PROGRAM S04_AluCovering
VAR
	//工站
	station					: REFERENCE TO FB_Station:=fbstation[4];
	//气缸
	fbHOZAdjustCyl_1	:REFERENCE TO FB_Cylinder:=fbCylinder[20];	//	上层水平调整气缸1
	fbHOZAdjustCyl_2	:REFERENCE TO FB_Cylinder:=fbCylinder[21];	//	上层水平调整气缸2
	fbHOZAdjustCyl_3	:REFERENCE TO FB_Cylinder:=fbCylinder[22];	//	下层水平调整气缸1
	fbHOZAdjustCyl_4	:REFERENCE TO FB_Cylinder:=fbCylinder[23];	//	下层水平调整气缸2
	//伺服
	fbZAxisMove_1	 :REFERENCE TO FB_Axis:=fbAxis[10];	//	热熔工位-Z轴伺服1（右）
	fbZAxisMove_2	 :REFERENCE TO FB_Axis:=fbAxis[11];	//		热熔工位-Z轴伺服2
	//温控器
	fbThermostat_1			 :REFERENCE TO FB_TempControl_FUSHI:=fbTempretureControl[1];//温控器1
    fbThermostat_2			 :REFERENCE TO FB_TempControl_FUSHI:=fbTempretureControl[2];//温控器2
	//延时
	arTonDelay :ARRAY[1..20] OF TON;
	//返回值
	UdiReturnValue :ARRAY[1..20] OF UDINT;
	//本地过程数据
	arProcessDataStation : ARRAY [1..2] OF DUT_MainlineFixture;
	i: INT;
	//过程记录
	tsModuleProcess:ARRAY[1..gc_ModuleProNo] OF DUT_Process;
	xClearModuleProcessDone:BOOL;
	bClearProcessStep	:BYTE;
END_VAR

ACTION A_Input:
//气缸
fbHOZAdjustCyl_1.xWP_Sensor	:=	IxS04HOZAdjustCyl_1WP	;
fbHOZAdjustCyl_1.xHP_Sensor	:=	IxS04HOZAdjustCyl_1HP	;
fbHOZAdjustCyl_2.xWP_Sensor	:=	IxS04HOZAdjustCyl_2WP	;
fbHOZAdjustCyl_2.xHP_Sensor	:=	IxS04HOZAdjustCyl_2HP	;
fbHOZAdjustCyl_3.xWP_Sensor	:=	IxS04HOZAdjustCyl_3WP	;
fbHOZAdjustCyl_3.xHP_Sensor	:=	IxS04HOZAdjustCyl_3HP	;
fbHOZAdjustCyl_4.xWP_Sensor	:=	IxS04HOZAdjustCyl_4WP	;
fbHOZAdjustCyl_4.xHP_Sensor	:=	IxS04HOZAdjustCyl_4HP	;
END_ACTION

ACTION Alarm:
//
station.adwAlarm[1].00:=station.xInitTimeout;	  			//S08Label 初始化超时
END_ACTION

ACTION Delay:
(*arTonDelay[01](IN:= , PT:=T#0.1S , Q=> , ET=> );*)//TipAuto使用
arTonDelay[02](IN:=  , PT:=stData.Thermostat[1].tTON_Delay , Q=> , ET=> );//热熔延时时间
arTonDelay[03](IN:=   , PT:=T#1S , Q=> , ET=> );
arTonDelay[04](IN:= , PT:=T#0.1S , Q=> , ET=> );
arTonDelay[05](IN:= , PT:=T#0.1S , Q=> , ET=> );
arTonDelay[06](IN:= , PT:=T#0.1S , Q=> , ET=> );
arTonDelay[07](IN:= , PT:=T#0.1S , Q=> , ET=> );
arTonDelay[08](IN:= , PT:=T#0.1S , Q=> , ET=> );
arTonDelay[09](IN:= , PT:=T#0.1S , Q=> , ET=> );
END_ACTION

ACTION FlowAuto:

//-----------------------------------------初始化是否完成判断----------------------------------------------
IF NOT station.xInitDone 
THEN
 	station.iStepAuto:=0;
 	station.xDone:=FALSE;
	station.xRunningOffProhibit := FALSE ;//运行中信号Off禁止
ELSIF station.xRunning  OR   tsModuleProcess[2].xProcessStarted
THEN
//-----------------------------------------动作步骤--------------------------------------------------------
CASE station.iStepAuto OF	  
	0: //----Home Step，等待启动----
		IF station.xDisabled 
			AND station.xCanRun 
			AND NOT fbMachine[1].xStopped 
			AND NOT station.xSingleRunning 
		THEN
			station.xDone:=TRUE;
		END_IF
		
		IF  station.xSingleRunning 
			OR station.xCanRun 
			AND NOT station.xDone 
			AND NOT station.xDisabled 
			AND NOT fbMachine[1].xStopped
		THEN
			station.xCycleEnable:=TRUE;
			station.xDone:= FALSE;  
			station.xRunningOffProhibit := TRUE ;//运行中信号Off禁止
			station.iStepAuto:= 10;
		END_IF
    10: //复位数据
			(*开启控温系统*) 
			fbThermostat_1.xStart :=TRUE;
			fbThermostat_2.xStart :=TRUE;
			arTonDelay[02](IN:= FALSE);
			station.iStepAuto:=20;	
	20:////Restore_after_Estop_Process1 上载数据流程
			IF  station.xSingleRunning OR  fbMachine[1].xTryRun THEN
					station.iStepAuto:=50;
			ELSIF tsModuleProcess[1].xProcessNotStarted AND NOT  tsModuleProcess[1].xProcessStarted THEN
					station.iStepAuto :=21; (*process not started*)
			ELSIF  tsModuleProcess[1].xProcessStarted AND NOT  tsModuleProcess[1].xProcessCompleted THEN
				 station.iStepAuto := 21;(*process started*)
			ELSIF  tsModuleProcess[1].xProcessCompleted AND NOT tsModuleProcess[1].xQDataCompleted  THEN
					station.iStepAuto := 40 ;(*process completed*)
			ELSIF tsModuleProcess[1].xQDataCompleted THEN
					station.iStepAuto :=40;(*Qdata completed *)
			ELSE
					station.iStepAuto :=21; 
			END_IF	
	21://
				tsModuleProcess[1].xProcessNotStarted:=TRUE;
				station.iStepAuto:= 30;
				
	30://数据load 
		tsModuleProcess[1].xProcessStarted	:=TRUE;
		MEMCPY(ADR(arProcessDataStation[1]),ADR(arMainlineFixtureData[arCurFixtureNumStation[10]]),SIZEOF(arMainlineFixtureData[arCurFixtureNumStation[10]]));
		MEMCPY(ADR(arProcessDataStation[2]),ADR(arMainlineFixtureData[arCurFixtureNumStation[11]]),SIZEOF(arMainlineFixtureData[arCurFixtureNumStation[11]]));
		tsModuleProcess[1].xProcessCompleted:=TRUE;
		tsModuleProcess[1].xQDataCompleted:=TRUE;
		station.iStepAuto:= 40;
	40: //判断产品状态
			IF  arProcessDataStation[1].xMaterialOnOff   AND
				 arProcessDataStation[2].xMaterialOnOff  THEN
				station.iStepAuto:= 41;
			ELSE
				station.iStepAuto:= 999;
			END_IF
	41://手动NOK按钮
			IF   arManualNOKHmiButton[4]  AND NOT station.xCycleRunning THEN
				station.iStepAuto:= 140;
			ELSE	
				station.iStepAuto:= 50;
			END_IF	
	
	/////产品流程开始	
	50:////Restore_after_Estop_Process2 热熔流程
			IF  station.xSingleRunning OR fbMachine[1].xTryRun THEN
					station.iStepAuto :=60; 
			ELSIF tsModuleProcess[2].xProcessNotStarted AND NOT  tsModuleProcess[2].xProcessStarted THEN
					station.iStepAuto :=60; (*process not started*)
			ELSIF  tsModuleProcess[2].xProcessStarted AND NOT  tsModuleProcess[2].xProcessCompleted THEN
				 station.iStepAuto := 140;(*process started*)
			ELSIF  tsModuleProcess[2].xProcessCompleted AND NOT tsModuleProcess[2].xQDataCompleted  THEN
					station.iStepAuto :=130;(*process completed*)
			ELSIF tsModuleProcess[2].xQDataCompleted THEN
					station.iStepAuto :=160;(*Qdata completed *)
			ELSE
					station.iStepAuto :=60; 
			END_IF	
	60://
				 tsModuleProcess[2].xProcessNotStarted:=TRUE;
				 station.iStepAuto :=70; 
	70://水平调整气缸伸出
					IF  iBoxChoose =1 THEN
						(*上层水平调整气缸*)
						fbHOZAdjustCyl_1.xAuto :=TRUE;
						fbHOZAdjustCyl_2.xAuto :=TRUE;
						IF  fbHOZAdjustCyl_1.xWP_Delay AND fbHOZAdjustCyl_2.xWP_Delay  THEN
								station.iStepAuto:= 80;
						END_IF
					ELSIF  iBoxChoose= 2 THEN
						(*下层水平调整气缸*)
						fbHOZAdjustCyl_3.xAuto :=TRUE;
						fbHOZAdjustCyl_4.xAuto :=TRUE;
						IF  fbHOZAdjustCyl_3.xWP_Delay AND fbHOZAdjustCyl_4.xWP_Delay  THEN
								station.iStepAuto:= 80;
						END_IF
					END_IF
	
	80://判断加热棒是否准备就绪
			IF  ( fbThermostat_1.xRdy AND  fbThermostat_2.xRdy ) OR 
				axBypassSignal[4] OR  fbMachine[1].xTryRun THEN
					station.iStepAuto:= 90;
			END_IF
	90://Z轴伺服下降到位置1
			tsModuleProcess[2].xProcessStarted:=TRUE;
			fbZAxisMove_1.xMoveAuto[2]:=TRUE;
			fbZAxisMove_2.xMoveAuto[2]:=TRUE;
			IF  fbZAxisMove_1.xMoveInPos[2] AND fbZAxisMove_2.xMoveInPos[2]THEN
				station.iStepInit:=100;	
			END_IF
	100://复位热熔时间
			arTonDelay[02](IN:=FALSE  , PT:=stData.Thermostat[1].tTON_Delay , Q=> , ET=> );//热熔延时时间
			station.iStepAuto:=110;
 	110://延时等待热熔完成
			arTonDelay[02](IN:=  , PT:=stData.Thermostat[1].tTON_Delay , Q=> , ET=> );//热熔延时时间
		IF  arTonDelay[02].Q  OR axBypassSignal[4]  OR fbMachine[1].xTryRun  THEN
			station.iStepInit:=120;	
			arTonDelay[02](IN:= FALSE );//热熔延时时间
		END_IF
	120://
			tsModuleProcess[2].xProcessCompleted :=TRUE;
			station.iStepInit:=130;	
	130://结果OK
			arProcessDataStation[1].stProduct.xAluCovering_NOK:=TRUE;
			arProcessDataStation[2].stProduct.xAluCovering_OK:=FALSE;
			station.iStepInit:=150;	
	140://结果NG 
			arProcessDataStation[1].stProduct.xAluCovering_NOK:=FALSE;
			arProcessDataStation[2].stProduct.xAluCovering_OK:=TRUE;		
			station.iStepInit:=150;	
	150:
			tsModuleProcess[2].xQDataCompleted :=TRUE;
			station.iStepInit:=160;	
	160://Z轴上升
			fbZAxisMove_1.xMoveAuto[1]:=TRUE;
			fbZAxisMove_2.xMoveAuto[1]:=TRUE;
			IF  fbZAxisMove_1.xMoveInPos[1] AND fbZAxisMove_2.xMoveInPos[1]THEN
				station.iStepInit:=170;	
			END_IF
	170://水平调整气缸收回
			fbHOZAdjustCyl_1.xAuto :=FALSE;
			fbHOZAdjustCyl_2.xAuto :=false;
			fbHOZAdjustCyl_3.xAuto :=false;
			fbHOZAdjustCyl_4.xAuto :=false;
		IF	fbHOZAdjustCyl_1.xhp_Delay AND
		    fbHOZAdjustCyl_2.xhp_Delay and
		    fbHOZAdjustCyl_3.xhp_Delay and
		    fbHOZAdjustCyl_4.xhp_Delay THEN
			station.iStepInit:=200;	
		END_IF
	////产品流程结束	
	200:////Restore_after_Estop_Process3 数据传输流程
			IF  station.xSingleRunning OR fbMachine[1].xTryRun THEN
					station.iStepAuto :=999; 
			ELSIF tsModuleProcess[3].xProcessNotStarted AND NOT  tsModuleProcess[3].xProcessStarted THEN
					station.iStepAuto :=210; (*process not started*)
			ELSIF  tsModuleProcess[3].xProcessStarted AND NOT  tsModuleProcess[3].xProcessCompleted THEN
				 station.iStepAuto := 220;(*process started*)
			ELSIF  tsModuleProcess[3].xProcessCompleted AND NOT tsModuleProcess[3].xQDataCompleted  THEN
					station.iStepAuto :=230;(*process completed*)
			ELSIF tsModuleProcess[3].xQDataCompleted THEN
					station.iStepAuto :=999;(*Qdata completed *)
			ELSE
					station.iStepAuto :=210; 
			END_IF		
	210://		
				tsModuleProcess[3].xProcessNotStarted:=TRUE;
				station.iStepAuto :=220; 
	220://数据unload
		tsModuleProcess[3].xProcessStarted:=TRUE;
		MEMCPY(ADR(arMainlineFixtureData[arCurFixtureNumStation[10]]),ADR(arProcessDataStation[1]),SIZEOF(arProcessDataStation[1]));
		MEMCPY(ADR(arMainlineFixtureData[arCurFixtureNumStation[11]]),ADR(arProcessDataStation[2]),SIZEOF(arProcessDataStation[2]));
		station.iStepAuto:= 230;
	230://
			tsModuleProcess[3].xProcessCompleted:=TRUE;
			station.iStepAuto :=240; 
 	240://本地数据清除
			MEMSET(ADR(arProcessDataStation[1]),0,SIZEOF(arProcessDataStation[1]));
			MEMSET(ADR(arProcessDataStation[2]),0,SIZEOF(arProcessDataStation[2]));
			arManualNOKHmiButton[4]:=FALSE;
			tsModuleProcess[3].xQDataCompleted:=TRUE;
			station.iStepAuto:= 999;
	999://----Single Run Finish----
			
		station.iStepAuto :=0;
		IF NOT station.xSingleContinuousRun THEN
			station.xSingleRunFlag:=FALSE;
		END_IF
		station.xCycleEnable:=FALSE;	
		station.xDone:=TRUE;
	ELSE
		;	
END_CASE



END_IF
END_ACTION

ACTION FlowInit:
IF NOT station.xIniting THEN
  station.iStepInit:=0;    
ELSE
//--------------------------------------------初始化步序----------------------------------
CASE station.iStepInit OF	
 0://  
  	IF station.xIniting THEN	
  	  station.iStepInit:=10;	
  	END_IF	
10://复位数据
	 station.iStepInit:=20;	
20://关闭控温系统
	fbThermostat_1.xStart :=FALSE;
	fbThermostat_2.xStart :=FALSE;
	 station.iStepInit:=30;	
30://Z轴伺服上电
	fbZAxisMove_1.xPowerInit:=TRUE;
    fbZAxisMove_2.xPowerInit:=TRUE;
	IF  fbZAxisMove_1.xPowerOn AND fbZAxisMove_2.xPowerOn THEN
		station.iStepInit:=40;	
	END_IF
40://Z轴伺服上升
	fbZAxisMove_1.xMoveAuto[1]:=TRUE;
    fbZAxisMove_2.xMoveAuto[1]:=TRUE;
	IF  fbZAxisMove_1.xMoveInPos[1] AND fbZAxisMove_2.xMoveInPos[1]THEN
		station.iStepInit:=50;	
	END_IF
50://水平调整气缸收回
	fbHOZAdjustCyl_1.xinit:=TRUE;	
	fbHOZAdjustCyl_2.xinit:=true;	
	fbHOZAdjustCyl_3.xinit:=true;	
	fbHOZAdjustCyl_4.xinit:=true;		
	IF     fbHOZAdjustCyl_1.xHp_Delay  AND 
		   fbHOZAdjustCyl_2.xHp_Delay  AND 
	 	   fbHOZAdjustCyl_3.xHp_Delay  AND 
           fbHOZAdjustCyl_4.xHp_Delay  THEN
			station.iStepInit:=100;
	END_IF
100://	
    station.iStepInit:=999;	
999://初始化完成	
	station.iStepInit:=0;
	station.xInitDone:=TRUE;  
END_CASE
END_IF
END_ACTION

ACTION General:
(******************清除过程记录**********************)
CASE bClearProcessStep OF
	0:	
		IF	 S08_MainLine.xClearProcessStatus THEN
			FOR i:=1 TO gc_ModuleProNo BY 1 DO
				MEMSET(ADR(tsModuleProcess[i]),0,SIZEOF(tsModuleProcess[i]));
			END_FOR
			bClearProcessStep:=10;
		END_IF
	10:
		xClearModuleProcessDone:=TRUE;
		bClearProcessStep:=20;
	20:
		IF NOT S08_MainLine.xClearProcessStatus THEN
			xClearModuleProcessDone:=FALSE;
			bClearProcessStep:=30;
		END_IF
	30:  
			bClearProcessStep:=0;
	
END_CASE
END_ACTION

ACTION ILC:

//---------------------------------------------------工站可执行-------------------------------------------------------
station.xCanRun :=TRUE ;

//---------------------------------------------------气缸动作条件-------------------------------------------
fbHOZAdjustCyl_1.xOffILC	:=	TRUE	;
fbHOZAdjustCyl_1.xOnILC	:=	TRUE	;
fbHOZAdjustCyl_2.xOffILC	:=	TRUE	;
fbHOZAdjustCyl_2.xOnILC	:=	TRUE	;
fbHOZAdjustCyl_3.xOffILC	:=	TRUE	;
fbHOZAdjustCyl_3.xOnILC	:=	TRUE	;
fbHOZAdjustCyl_4.xOffILC	:=	TRUE	;
fbHOZAdjustCyl_4.xOnILC	:=	TRUE	;


//---------------------------------------------------伺服动作条件-------------------------------------------

fbZAxisMove_1.xRunILC := 
fbZAxisMove_1.xMoveILC[1] :=
fbZAxisMove_1.xMoveILC[2] :=
fbZAxisMove_1.xMoveILC[3] :=
fbZAxisMove_1.xMoveILC[4] :=
fbZAxisMove_1.xMoveILC[5] := TRUE ;

fbZAxisMove_2.xRunILC := 
fbZAxisMove_2.xMoveILC[1] :=
fbZAxisMove_2.xMoveILC[2] :=
fbZAxisMove_2.xMoveILC[3] :=
fbZAxisMove_2.xMoveILC[4] :=
fbZAxisMove_2.xMoveILC[5] := TRUE ;
END_ACTION

ACTION TipAuto:

//------------------------------------------------AutoTip Cylinder--------------------------------
station.adwAutoTip[1].00	:=	fbHOZAdjustCyl_1.xAutoTip	;
station.adwAutoTip[1].01	:=	fbHOZAdjustCyl_2.xAutoTip	;
station.adwAutoTip[1].02	:=	fbHOZAdjustCyl_3.xAutoTip	;
station.adwAutoTip[1].03	:=	fbHOZAdjustCyl_4.xAutoTip	;
	
//------------------------------------------------AutoTip Servo--------------------------------
//**************************************
FOR i:= 1 TO 5 BY 1 DO 
	IF fbZAxisMove_1.xMoveAuto[i] THEN
		fbZAxisMove_1.iPosNumber := i ;
	END_IF
	IF fbZAxisMove_2.xMoveAuto[i] THEN
		fbZAxisMove_2.iPosNumber := i ;
	END_IF
	
END_FOR

IF  fbMachine[1].xAutoMode AND NOT fbMachine[1].xRunning  THEN
	  arTonDelay[01](IN:=True , PT:=T#1S , Q=> , ET=> );
else
	  arTonDelay[01](IN:=false);
END_IF
IF arTonDelay[1].Q  THEN 
	IF	fbZAxisMove_1.iPosNumber=1 	AND NOT fbZAxisMove_1.xMoveInPos[1] 	THEN 	station.adwAutoTip[1].10:=TRUE	;	END_IF//轴伺服自动时位置不在位置1
	if	fbZAxisMove_1.iPosNumber=2	AND NOT fbZAxisMove_1.xMoveInPos[2]	THEN 	station.adwAutoTip[1].11:=TRUE	;	END_IF//轴伺服自动时位置不在位置2
	if	fbZAxisMove_1.iPosNumber=3	AND NOT fbZAxisMove_1.xMoveInPos[3]	THEN 	station.adwAutoTip[1].12:=TRUE	;	END_IF//轴伺服自动时位置不在位置3
	if	fbZAxisMove_1.iPosNumber=4	AND NOT fbZAxisMove_1.xMoveInPos[4]	THEN 	station.adwAutoTip[1].13:=TRUE	;	END_IF//轴伺服自动时位置不在位置4
	if	fbZAxisMove_1.iPosNumber=5	AND NOT fbZAxisMove_1.xMoveInPos[5]	THEN 	station.adwAutoTip[1].14:=TRUE	;	END_IF//轴伺服自动时位置不在位置5
	IF	fbZAxisMove_2.iPosNumber=1 	AND NOT fbZAxisMove_2.xMoveInPos[1] 	THEN 	station.adwAutoTip[1].15:=TRUE	;	END_IF//轴伺服自动时位置不在位置1
	if	fbZAxisMove_2.iPosNumber=2	AND NOT fbZAxisMove_2.xMoveInPos[2]	THEN 	station.adwAutoTip[1].16:=TRUE	;	END_IF//轴伺服自动时位置不在位置2
	if	fbZAxisMove_2.iPosNumber=3	AND NOT fbZAxisMove_2.xMoveInPos[3]	THEN 	station.adwAutoTip[1].17:=TRUE	;	END_IF//轴伺服自动时位置不在位置3
	if	fbZAxisMove_2.iPosNumber=4	AND NOT fbZAxisMove_2.xMoveInPos[4]	THEN 	station.adwAutoTip[1].18:=TRUE	;	END_IF//轴伺服自动时位置不在位置4
	if	fbZAxisMove_2.iPosNumber=5	AND NOT fbZAxisMove_2.xMoveInPos[5]	THEN 	station.adwAutoTip[1].19:=TRUE	;	END_IF//轴伺服自动时位置不在位置5
	
	
		
END_IF
END_ACTION

ACTION TipManual:
//--------------------------------------------ManualTip------------------------------------------------------

//-------------------------------------------气缸提示---------------------------------------------------------




/////////////////////////////////////////////////////////////////////////////////////////////////////////////////
END_ACTION

ACTION Z_Output:
(**************************气缸输出********************************)
QxS04HOZAdjustCyl_1WP	:=	fbHOZAdjustCyl_1.xWP_Valve	;
QxS04HOZAdjustCyl_1HP	:=	fbHOZAdjustCyl_1.xHP_Valve	;
QxS04HOZAdjustCyl_2WP	:=	fbHOZAdjustCyl_2.xWP_Valve	;
QxS04HOZAdjustCyl_2HP	:=	fbHOZAdjustCyl_2.xHP_Valve	;
QxS04HOZAdjustCyl_3WP	:=	fbHOZAdjustCyl_3.xWP_Valve	;
QxS04HOZAdjustCyl_3HP	:=	fbHOZAdjustCyl_3.xHP_Valve	;
QxS04HOZAdjustCyl_4WP	:=	fbHOZAdjustCyl_4.xWP_Valve	;
QxS04HOZAdjustCyl_4HP	:=	fbHOZAdjustCyl_4.xHP_Valve	;
END_ACTION

END_PROGRAM

(* stored: Version 1.1.0.1, ProductVersion 3.1.4024.9
   POU S04_AluCovering: Id {9f04510a-7cb9-4290-b624-ad41194a4509}, SpecialFunc None
   Action A_Input: Id {65b47811-5915-4744-a63e-96ca1ba2a959}
   Action Alarm: Id {4b5e4421-5305-4405-b11b-0af4cd39b3da}
   Action Delay: Id {26e43c03-7b70-412e-9d66-6498126722fc}
   Action FlowAuto: Id {e3e998e8-11c4-417d-bceb-b9a63717ba8e}
   Action FlowInit: Id {064317f4-3489-452e-ac7f-03fe87bc3d78}
   Action General: Id {81d8e462-a9d5-4975-910b-41bf7bc2abe3}
   Action ILC: Id {093b9242-4feb-4df4-b145-2493df43265e}
   Action TipAuto: Id {8e1c36ee-890f-4b23-a358-969bda10a9be}
   Action TipManual: Id {4fcf71f6-e5c5-4ba5-9691-e06d4cc0f64f}
   Action Z_Output: Id {9e3423bb-d549-4f1c-bdf2-1776371802b4} *)
